{attribute 'qualified_only'}
{attribute 'strict'}
TYPE E_EquipmentUpdate :
(
	Manual := 1,
	Auto := 2,
	Offline := 3,
	Running := 4,
	SleepActive := 5,
	Faulted := 6,
	OverHeight := 7
);
END_TYPE

(* stored: Version 1.1.0.1, ProductVersion 3.1.4024.4
   EnumerationTextList E_EquipmentUpdate: Id {718c5326-ae2f-4bec-9265-901f9d721783} *)
